FUNCTION_BLOCK FB_Ethercat EXTENDS FB_Component
VAR_INPUT
    NetId 			AT %I*:		T_AmsNetIdArr;
END_VAR
VAR_OUTPUT
END_VAR
VAR
	sNetId:						T_AmsNetID;
	nSlaves:					UINT;
	fbGetMasterState: 			FB_EcGetMasterDevState;
	fbGetSlaveStates:			FB_EcGetAllSlaveStates;
	fbGetConfSlaves: 			FB_EcGetConfSlaves;
	fbGetSlaveCount:			FB_EcGetSlaveCount;
	fbGetSlaveAddresses:		FB_EcGetAllSlaveAddr;
END_VAR

METHOD FB_exit : BOOL
VAR_INPUT
	bInCopyCode : BOOL; // if TRUE, the exit method is called for exiting an instance that is copied afterwards (online change).
END_VAR
IF fbGetSlaveStates.pStateBuf <> 0 THEN
	__DELETE(fbGetSlaveStates.pStateBuf);
END_IF
IF fbGetConfSlaves.pArrEcConfSlaveInfo <> 0 THEN
	__DELETE(fbGetConfSlaves.pArrEcConfSlaveInfo);
END_IF
END_METHOD

METHOD PROTECTED M_Execute : BOOL // Return state complete
VAR_INPUT
END_VAR
VAR
	nIndex:					UINT;
END_VAR
fbGetMasterState(bExecute:= NOT fbGetMasterState.bBusy);
IF fbGetMasterState.bError THEN
	fbEvent.M_Abort('Ethercat master state', '');
END_IF

fbGetSlaveStates(bExecute:= NOT fbGetSlaveStates.bBusy);

FOR nIndex:= 0 TO fbGetSlaveStates.nSlaves -1 DO
	CASE fbGetSlaveStates.pStateBuf^[nIndex].deviceState OF
		EC_DEVICE_STATE_INIT:;
		EC_DEVICE_STATE_PREOP:;
		EC_DEVICE_STATE_BOOTSTRAP:;
		EC_DEVICE_STATE_SAFEOP:;
		EC_DEVICE_STATE_OP:;
	END_CASE
END_FOR

fbGetSlaveAddresses(bExecute:= TRUE);

fbGetConfSlaves(bExecute:= TRUE);
END_METHOD

METHOD PROTECTED M_Starting : BOOL // Return state complete
VAR_INPUT
END_VAR
VAR
END_VAR

sNetId:= F_CreateAmsNetId(NetId);

IF F_GetMappingStatus(ADR(NetId), SIZEOF(T_AmsNetIdArr)) <> EPlcMappingStatus.MS_Mapped THEN
	fbEvent.M_AddSTRING(sNetId);
	fbEvent.M_Abort('Ethercat master netid not mapped %s', '');
END_IF

fbGetMasterState.sNetId:= sNetId;
fbGetSlaveAddresses.sNetId:= sNetId;
fbGetSlaveStates.sNetId:= sNetId;
fbGetConfSlaves.sNetId:= sNetId;

fbGetSlaveCount.sNetId:= sNetId;
fbGetSlaveCount(bExecute:= TRUE);
IF NOT fbGetSlaveCount.bBusy THEN
	nSlaves:= fbGetSlaveCount.nSlaves;
	
		IF fbGetSlaveStates.pStateBuf = 0 THEN
			IF fbGetSlaveStates.cbBufLen <> 0 THEN
				__DELETE(fbGetSlaveStates.pStateBuf);
			END_IF
			fbGetSlaveStates.cbBufLen:= nSlaves * SIZEOF(Tc2_EtherCAT.ST_EcSlaveState);
			fbGetSlaveStates.pStateBuf:= __NEW(BYTE, fbGetSlaveStates.cbBufLen); 	
		END_IF
		
		IF fbGetConfSlaves.pArrEcConfSlaveInfo = 0 THEN
			IF fbGetConfSlaves.pArrEcConfSlaveInfo <> 0 THEN
				__DELETE(fbGetConfSlaves.pArrEcConfSlaveInfo);
			END_IF
			fbGetConfSlaves.cbBufLen:= nSlaves * SIZEOF(Tc2_EtherCAT.ST_EcSlaveConfigData);
			fbGetConfSlaves.pArrEcConfSlaveInfo:=  __NEW(BYTE, fbGetConfSlaves.cbBufLen);

		END_IF
		
		IF fbGetSlaveAddresses.pAddrBuf = 0 THEN
			IF fbGetSlaveAddresses.pAddrBuf <> 0 THEN
				__DELETE(fbGetSlaveAddresses.pAddrBuf);
			END_IF
			fbGetSlaveAddresses.cbBufLen:= nSlaves * SIZEOF(UINT);
			fbGetSlaveAddresses.pAddrBuf:=  __NEW(BYTE, fbGetSlaveAddresses.cbBufLen);
		END_IF	

	M_Starting:= TRUE;
END_IF
END_METHOD

END_FUNCTION_BLOCK

(* stored: Version 1.1.0.1, ProductVersion 3.1.4024.12
   POU FB_Ethercat: Id {26632774-44df-0f9a-1531-badc4b6ed605}, SpecialFunc None
   Method FB_exit: Id {32b88d2f-9681-0500-1b45-7ff197d7c043}
   Method M_Execute: Id {2ba98b6e-4256-0860-0cd0-bd9578cd5e7c}
   Method M_Starting: Id {429ce4f6-d8ad-000d-1883-5a642980062d} *)
